// TIA Portal project "RedArrowMQTT" (V15)

(* hardware
DEVICE "S7-1200 station_1"  S7-1200 Station
   slot 0: "Rack_0"  S7-1200 Rack  Rack  V1.0
   slot 1: "PLC_1"  CPU 1214C AC/DC/Rly  6ES7 214-1BG40-0XB0  V4.2
*)

// ===== PLC "PLC_1"  CPU 1214C AC/DC/Rly =====

VAR_GLOBAL   // PLC tag table "Default tag table"
   "System_Byte" AT %MB1 : Byte;
   "FirstScan" AT %M1.0 : Bool;
   "DiagStatusUpdate" AT %M1.1 : Bool;
   "AlwaysTRUE" AT %M1.2 : Bool;
   "AlwaysFALSE" AT %M1.3 : Bool;
   "Clock_Byte" AT %MB0 : Byte;
   "Clock_10Hz" AT %M0.0 : Bool;
   "Clock_5Hz" AT %M0.1 : Bool;
   "Clock_2.5Hz" AT %M0.2 : Bool;
   "Clock_2Hz" AT %M0.3 : Bool;
   "Clock_1.25Hz" AT %M0.4 : Bool;
   "Clock_1Hz" AT %M0.5 : Bool;
   "Clock_0.625Hz" AT %M0.6 : Bool;
   "Clock_0.5Hz" AT %M0.7 : Bool;
   "miState" AT %MW50 : Int;
   "miCurrentLocation" AT %MW52 : Int;
   "SerializeResult" AT %MW56 : Int;
   "charCount" AT %MW54 : Int;
   "bSendMessage" AT %M35.0 : Bool;
   "bSubscribe" AT %M35.1 : Bool;
END_VAR

VAR_GLOBAL CONSTANT   // PLC tag table "IOT Constants"
   "ciSubMessageReceived" : Int := 15;
   "ciDisablePublish" : Int := 0;
   "ciSubReadyToSub" : Int := 10;
   "ciSubDisabled" : Int := 0;
   "ciSubSubscribed" : Int := 20;
   "ciReadyToPublish" : Int := 10;
END_VAR

VAR_GLOBAL CONSTANT   // PLC tag table "MQTT Message Constants"
   "ciRemovalRequested" : Int := 2;
   "ciAdditionRequested" : Int := 1;
   "ciDriverIDLength" : Int := 8;
   "ciVehicleIDLength" : Int := 8;
   "ciCustomerNameLength" : Int := 20;
   "ciMaxDrivers" : Int := 1000;
   "ciMaxVehicles" : Int := 1000;
   "ciMaxCustomers" : Int := 5;
   "ciWashesPerVehicle" : Int := 5;
   "ciSyncBufferSize" : Int := 75;
   "ciVersionNumber" : String := '/V3';
   "ciCustomerSyncBufferSize" : Int := 5;
END_VAR

TYPE "udtDriver"
   STRUCT
      sDriverID : String["ciDriverIDLength"];   // Driver's alphanumeric ID
      iCustomer : USInt;   // Index of customer to which driver belongs
   END_STRUCT;
END_TYPE

TYPE "udtVehicle"
   STRUCT
      sVehicleID : String["ciVehicleIDLength"];   // Vehicle ID
      iWashesAvailable : Array[1.."ciWashesPerVehicle"] of USInt;   // Set of wash types available to this vehicle
      iCustomer : USInt;   // Index of customer to which vehicle belongs
   END_STRUCT;
END_TYPE

TYPE "udtUserList"
   STRUCT
      Drivers : Array[1.."ciMaxDrivers"] of "udtDriver";
      Vehicles : Array[1.."ciMaxVehicles"] of "udtVehicle";
      Customers : Array[1.."ciMaxCustomers"] of String[20];
      sCurrentDriver : String["ciDriverIDLength"];
      sCurrentVehicleID : String["ciVehicleIDLength"];
      iCurrentWashesAvailable : Array[1.."ciWashesPerVehicle"] of USInt;
      iCurrentCustomer : USInt;
      sCurrentCustomerName : String["ciCustomerNameLength"];
   END_STRUCT;
END_TYPE

TYPE "udtError_Drivers"
   STRUCT
      DriverOverfill : Bool;   // Driver cannot be added because queue is full
      DriverDoesNotExist : Bool;   // Driver cannot be removed because they do not exist
      DriverExists : Bool;   // Driver cannot be added because they already exist
      CustomerDoesNotExist : Bool;   // Driver cannot be added or removed because customer does not exist
      SyncBufferOverfill : Bool;   // Sync operation cannot be completed due to lack of space
   END_STRUCT;
END_TYPE

TYPE "udtError_Vehicles"
   STRUCT
      VehicleOverfill : Bool;   // Vehicle cannot be added because queue is full
      VehicleDoesNotExist : Bool;   // Vehicle cannot be removed because they do not exist
      VehicleExists : Bool;   // Vehicle cannot be added because they already exist
      CustomerDoesNotExist : Bool;   // Vehicle cannot be added because customer does not exist
      SyncBufferOverfill : Bool;
   END_STRUCT;
END_TYPE

TYPE "udtError_Customer"
   STRUCT
      CustomerOverfill : Bool;   // Customer queue full
      CustomerAlreadyExists : Bool;   // Cannot add customer because they already exist
      CustomerDoesNotExist : Bool;   // Cannot remove custome because they do not exist
      SyncBufferOverfill : Bool;   // Customer sync buffer is full
   END_STRUCT;
END_TYPE

TYPE "udtCustomer"
   STRUCT
      sCustomerName : String["ciCustomerNameLength"];
      aVehicles : Array[1.."ciMaxVehicles"] of "udtVehicle";
      aDrivers : Array[1.."ciMaxDrivers"] of String["ciDriverIDLength"];
      Sync : Struct
         iTotalDrivers : Int;
         iTotalVehicles : Int;
         iDriversSynced : Int;   // Counter for how many drivers IDs have been sent so far suring the sync process
         iVehiclesSynced : Int;   // Counter for how many vehicles have been sent so far in the sync process
         sDriverSyncBuffer : Array[1.."ciSyncBufferSize"] of String[8];
         VehicleSyncBuffer : Array[1.."ciSyncBufferSize"] of "udtVehicle";
         bDriverSyncComplete : Bool;
         bVehicleSyncComplete : Bool;
         bDriverSync : Array[1.."ciMaxDrivers"] of Bool;   // Bit indicating if a driver at a given index has been synced
         bVehicleSync : Array[1.."ciMaxVehicles"] of Bool;   // Bit indicating if a vehicle at a given index has been synced
         bCustomerSync : Bool;
      END_STRUCT;
   END_STRUCT;
END_TYPE

TYPE "udtCustomerList"
   STRUCT
      aCustomers : Array[1.."ciMaxCustomers"] of "udtCustomer";
      sCurrentDriver : String["ciDriverIDLength"];
      sCurrentVehicleID : String["ciVehicleIDLength"];
      iCurrentWashesAvailable : Array[1.."ciWashesPerVehicle"] of USInt;
      iCurrentCustomer : USInt;
      sCurrentCustomerName : String["ciCustomerNameLength"];
      iTotalCustomers : Int;
      iCustomersSynced : Int;
   END_STRUCT;
END_TYPE

TYPE "udtWashReportRaw"
   STRUCT
      bInWashComplete : Bool := false;   // Trigger to start the serialization
      bInMaxRuntimeTripped : Bool;   // Set if the user wash in wash for more than max allowed time
      DTL_StartTime : DTL;   // Starting date and time of wash
      tInTotalTime : Time;   // Total time in wash
      iInWashType : USInt;   // Wash type ID
      tInArch1Time : Time;
      tInArch2Time : Time;
      tInArch3Time : Time;
      tInArch4Time : Time;
      tInArch5Time : Time;
   END_STRUCT;
END_TYPE

TYPE "udtWashReportSend"
   STRUCT
      sCustomer : String["ciCustomerNameLength"];   // Customer Name
      sDriverID : String["ciDriverIDLength"];   // 8 character alphanumeric driver ID
      sVehicleID : String["ciVehicleIDLength"];   // 8 character alphanumeric vehicle ID
      iWashType : UInt;   // Wash type received
      bInMaxRuntimeTripped : Bool;   // Set if the user wash in wash for more than max allowed time
      iYear : UInt;   // Year
      iMonth : UInt;   // Month
      iDay : UInt;   // Day
      iHour : UInt;   // Hour
      iMinute : UInt;   // Minute
      iSecond : UInt;   // Second
      iTotalTime : UInt;   // Total time in wash
      iArch1Time : UInt;   // Time under arch 1
      iArch2Time : UInt;   // Time under arch 2
      iArch3Time : UInt;   // Time under arch 3
      iArch4Time : UInt;   // Time under arch 4
      iArch5Time : UInt;   // Time under arch 5
   END_STRUCT;
END_TYPE

TYPE "udtSyncLog"
   STRUCT
      iTotalCustomers : UInt;
      iTotalDrivers : UInt;
      iTotalVehicles : UInt;
      iCustomersSynced : USInt;
      iVehiclesSynced : UInt;
      iDriversSynced : UInt;
      CustomerSyncBuffer : Array[1.."ciCustomerSyncBufferSize"] of String["ciCustomerNameLength"];
      DriverSyncBuffer : Array[1.."ciSyncBufferSize"] of "udtDriver";
      VehicleSyncBuffer : Array[1.."ciSyncBufferSize"] of "udtVehicle";
      bDriverSync : Array[1.."ciMaxDrivers"] of Bool;
      bVehicleSync : Array[1.."ciMaxVehicles"] of Bool;
      bCustomerSync : Array[1.."ciMaxCustomers"] of Bool;
   END_STRUCT;
END_TYPE

// folder: MQTT

TYPE "udtMQTT_SubcribeMessageBuffer"
   STRUCT
      Message : Array[1..20] of "udtMQTT_SubscribeMessage";   // udtMQTT_SubscribeMessage
   END_STRUCT;
END_TYPE

TYPE "udtMQTT_SubscribeMessage"
   STRUCT
      iStatus : Int;   // Message status
      iQoS : Int;   // Quality of service value (0 or 1)
      sTopic : String[75];   // Topic to which its subscribed
      byValue : Array[0..75] of Byte;   // Byte array of message contents
      iMessageLength : Int;   // Length of received message
   END_STRUCT;
END_TYPE

TYPE "udtMQTT_PublishMessage"
   STRUCT
      iStatus : Int;   // Message Status
      iQoS : Int;   // Quality of service value (0 or 1)
      sTopic : String;   // Topic of sent message
      byValue : Array[0..100] of Byte;   // Byte array of message contents
      iMessageLength : DInt;   // Length of byValue occupied by relevant data
   END_STRUCT;
END_TYPE

TYPE "udtMQTT_PublishMessageBuffer"
   STRUCT
      iIndexWrite : Int;   // Message index currently being written by an fcMQTT_SerializeMessage block
      iIndexMax : Int := 3;   // Max index writtable within the message array
      bErrorOverfill : Bool;   // Set when fcMQTT_SerializeMessage tries to write to an unsent message
      Message : Array[1..10] of "udtMQTT_PublishMessage";   // udtMQTT_PublishMessage
   END_STRUCT;
END_TYPE

TYPE "udtError_MQTT"
   STRUCT
      ConSendErr : Bool;
      ConSendTO : Bool;
      ConAckRcvErr : Bool;
      ConAckTO : Bool;
      ConAckIncReply : Bool;
      ConAckIncLen : Bool;
      ConAckUnacProt : Bool;
      ConAckIdRej : Bool;
      ConAckSerUn : Bool;
      ConAckUserPass : Bool;
      ConAckNotAut : Bool;
      ConAckUnknown : Bool;
      PubSendErr : Bool;
      PubSendTO : Bool;
      PubAckRcvErr : Bool;
      PubAckTO : Bool;
      PubAckIncReply : Bool;
      PubAckIncLen : Bool;
      PubAckPacketID : Bool;
      SubSendErr : Bool;
      SubSendTimeout : Bool;
      SubAckIncReply : Bool;
      SubAckPacketID : Bool;
      SubAckRcvErr : Bool;
      SubAckTO : Bool;
      SubTopicNotFound : Bool;
      SubSendPubAckErr : Bool;
      SubSendPubAckTO : Bool;
      TcpErr : Bool;
      TcpTO : Bool;
      QueueOverflow : Bool;
   END_STRUCT;
END_TYPE

// folder: (top level)

DATA_BLOCK "IOT Communication_DB"   // DB3
{ S7_Optimized_Access := 'TRUE' }
VERSION : 0.1
// stored: InstanceOfName IOT Communication
"IOT Communication"
BEGIN
END_DATA_BLOCK

DATA_BLOCK "fbMain_DB"   // DB4
{ S7_Optimized_Access := 'TRUE' }
VERSION : 0.1
// stored: InstanceOfName fbMain
"fbMain"
BEGIN
END_DATA_BLOCK

DATA_BLOCK "dbErrors"   // DB7
{ S7_Optimized_Access := 'TRUE' }
VERSION : 0.1
   VAR
      Error_MQTT : "udtError_MQTT";
      Error_Drivers : "udtError_Drivers";
      Error_Vehicles : "udtError_Vehicles";
      Error_Customers : "udtError_Customer";
   END_VAR
BEGIN
END_DATA_BLOCK

// folder: MQTT

DATA_BLOCK "dbMQTT_MessageBuffer"   // DB1
{ S7_Optimized_Access := 'TRUE' }
VERSION : 0.1
   VAR
      OutgoingMessages : "udtMQTT_PublishMessageBuffer";
      IncomingMessages : "udtMQTT_SubcribeMessageBuffer";
      ErrorMessages : "udtMQTT_PublishMessageBuffer";
   END_VAR
BEGIN
   OutgoingMessages.iIndexMax := 10;
   ErrorMessages.iIndexMax := 10;
   IncomingMessages.Message[1].iStatus := 0;
   IncomingMessages.Message[2].iStatus := 0;
   IncomingMessages.Message[3].iStatus := 0;
END_DATA_BLOCK

DATA_BLOCK "dbMQTT_Data"   // DB26
TITLE = gdbIOTData_V1
{ S7_Optimized_Access := 'FALSE' }
AUTHOR : Eric_Niebylski
VERSION : 0.1
// Added rTargetRate ro 10minDataorAlarm
   VAR
      TestTopic : Struct   // To IOT Only
         DeviceID : String[9] := 'Something';
      END_STRUCT;
      ConfigData : Struct   // Bi
         Param1 : Int;
         Param2 : Int;
         Param3 : Real;
      END_STRUCT;
      sTemp : String;
      testCharArray : Array[1..20] of Char;
      rTemp : Real;
      itemp : Int;
      wError : Word;
   END_VAR
BEGIN
END_DATA_BLOCK

// folder: System blocks/Program resources

DATA_BLOCK "MQTT_TCON_Param"   // DB2
{ S7_Optimized_Access := 'TRUE' }
AUTHOR : SIMATIC
FAMILY : MC7Plus
NAME : TCON_Prm
VERSION : 1.0
// stored: InstanceOfName TCON_Param
"TCON_Param"
BEGIN
   REM_TSAP_ID[1] := 16#07;
   REM_TSAP_ID[2] := 16#5B;
   ID := 4;
END_DATA_BLOCK

// folder: (top level)

FUNCTION_BLOCK "fbMain"   // FB1, LAD
{ S7_Optimized_Access := 'TRUE' }
VERSION : 0.1
   VAR
      ins_GET_IM_DATA : Get_IM_Data;
      IMData : IM0_Data;
      bIMDataDone : Bool;
      bReadyToSub : Bool;   // Ready to subscribe to topics
      insFb_TankLevel : "fbTankLevel";
      bInMid : Bool;
      bInLow : Bool;
      bValidDriver : Bool;
      bValidVehicle : Bool;
      "IOT Communication_DB" : "IOT Communication";
      bWashReportSend : Bool;
      TON_WashReportSend : TON_TIME;
   END_VAR
   VAR_TEMP
      iTemp1 : Int;
      diTemp : DInt;
      bTemp : Bool;
      wTemp : Word;
   END_VAR
BEGIN

REGION Network 1
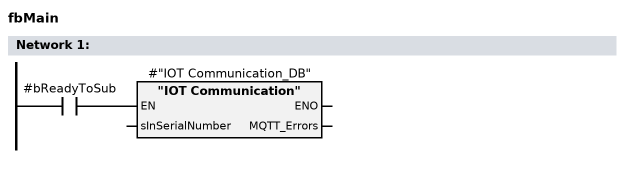
   RUNG wire#powerrail
      Contact( #bReadyToSub )
      #"IOT Communication_DB"(sInSerialNumber :=, MQTT_Errors =>)
   END_RUNG
   // the same network as SCL:
   IF #bReadyToSub THEN
       #"IOT Communication_DB"();   // "IOT Communication"
   END_IF;
END_REGION
END_FUNCTION_BLOCK

ORGANIZATION_BLOCK "Main"   // OB1, LAD, ProgramCycle
TITLE = "Main Program Sweep (Cycle)"
{ S7_Optimized_Access := 'TRUE' }
VERSION : 0.1
   VAR_INPUT
      Initial_Call : Bool;   // Initial call of this OB
      Remanence : Bool;   // =True, if remanent data are available
   END_VAR
BEGIN

REGION Network 1
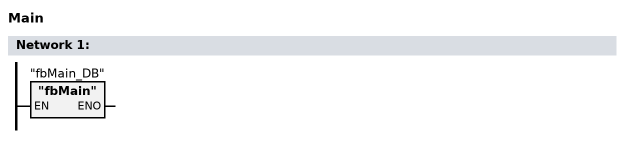
   RUNG wire#powerrail
      "fbMain_DB"()
   END_RUNG
   // the same network as SCL:
   "fbMain_DB"();   // "fbMain"
END_REGION
END_ORGANIZATION_BLOCK

// folder: MQTT

FUNCTION_BLOCK "IOT Communication"   // FB18, SCL
{ S7_Optimized_Access := 'TRUE' }
VERSION : 0.1
   VAR_INPUT
      sInSerialNumber : String;
   END_VAR
   VAR_OUTPUT
      MQTT_Errors : "udtError_MQTT";   // MQTT Error udt
   END_VAR
   VAR
      MQTT : "fbMQTT";
      bSerializeDone : Array[0..10] of Bool;
      bSerializeHold : Array[0..10] of Bool;
      bNewMessage : Array[0..10] of Bool;
      bInTankMidSensor : Bool;   // Temporary, replace with DI
      bInTankLowSensor : Bool;   // Temporary, replace with DI
      TankLevel : "fbTankLevel";
      bSendTankReport : Bool;
      iCustomersSynced : Int;
      sLastCustomerSync : String["ciCustomerNameLength"];
      sLastDriverSync : String["ciDriverIDLength"];
      sLastDriverCustomer : String["ciCustomerNameLength"];
      sLastVehicleSync : String["ciVehicleIDLength"];
      sLastVehicleCustomer : String["ciCustomerNameLength"];
   END_VAR
   VAR_TEMP
      tempTime : Time;
      bTemp : Bool;
      iIndex : Int;
      i : Int;
      diTemp : DInt;
   END_VAR
BEGIN
   // MQTT communication control driver
   #MQTT(sInClientID := 'ClientID',
         sInUserName := 'UserName',
                sInPassword := '12345',
                TCON_Param := "MQTT_TCON_Param",
                ERROR_MQTT := #MQTT_Errors);


    // Serialize message Structure to be sent
   "fcMQTT_SerializeMessageRaw"(sInSerial:=_string_in_,
                                sInTopic:=_string_in_,
                                sInVersion:=_string_in_,
                                iInQoS:=_int_in_,
                                Message:=_variant_in_,
                                bOutMessageSerialized=>_bool_out_);

   //Subscribe to message and send to DB
   "fcMQTT_DeserializeMessageSubscribe"(sInTopic:=_string_in_,
                                        iInQoS:=_int_in_,
                                        iInBufferIndex:=_int_in_,
                                        sInSerial:=_string_in_,
                                        sInVersion:=_string_in_,
                                        Message=>_variant_out_,
                                        bOutNewMessage=>_bool_out_);
END_FUNCTION_BLOCK

FUNCTION_BLOCK "fbMQTT"   // FB19, SCL
{ S7_Optimized_Access := 'TRUE' }
VERSION : 0.1
   VAR_INPUT
      sInClientID : String;   // Client ID, 23 char max / Client ID
      sInUserName : String;   // Username
      sInPassword : String;   // Password
      bInCleanSession : Bool;   // 0=Reuse prev session; 1=Discard prev sessions and start new one / Set high to clean session
      bInResetError : Bool;   // Error Reset
   END_VAR
   VAR_OUTPUT
      bOutError : Bool;   // Error present
   END_VAR
   VAR_IN_OUT
      ERROR_MQTT : "udtError_MQTT";   // Error udt
      TCON_Param : TCON_Param;   // Connection paramters
   END_VAR
   VAR
      iStatePublish : Int := 10;   // Current state of publish state machine
      iStateSubscribe : Int := 10;   // Current state of subscribe state machine
      iSelQueueIndexPublish : Int;   // Queue index of message currently being published
      iPrevSelQueueIndexPublish : Int;   // Queue index of last message to be published
      iPublishIndex : Int;   // Current byte index of message to be published
      uiSendLen : UInt;   // Length of message being sent
      uiPubPacketID : UInt;   // Unique ID for each sent packet
      bPubInProgress : Bool;   // Publication of packet in progress
      iSubscribeIndex : Int;   // Queue index of message whose topic is being subscribed to
      uiSubPacketID : UInt;   // ID of subcribe packet. Expected in suback packet.
      iSubMessageIndex : Int;   // Current byte of current working subscription related message
      bSubInProgress : Bool;   // Set if busy subscribing to a topic
      bSubReceiveInProgress : Bool;   // Set if busy receiving data on a subscribed topic
      iSubReceivedQoS : Int;   // QoS of received publish packet
      iReceivedTopicLength : Int;   // Length of a received topic (in bytes)
      sReceivedTopic : String;   // Topic of received message
      iTopicIndex : Int;   // Index of received topic within Incoming Messages
      bConAckReceived : Bool;   // Conack packet received
      bPubAckReceived : Bool;   // Puback packet received
      bSubAckReceived : Bool;   // Suback packet received
      bPublishReceived : Bool;   // Publish packet received
      iPayloadStartIndex : Int;   // Start index of payload of received publish packet
      iEndOfPayloadIndex : Int;   // End index of payload of received publish packet
      byData : Array[1..200] of Byte;   // Max: id+user+password+buffer
      byDataNewMessage : Array[1..300] of Byte;
      fbTCON : TCON;   // fb to establish TCP connection
      fbTDISCON : TDISCON;   // fb to disconnect from TCP
      fbTSEND : TSEND;   // fb for sending packets
      fbTRCV : TRCV;   // fb for receiving packets
      TON_TimeoutPub : TON_TIME;   // Publish timeout timer
      TON_TimeoutSub : TON_TIME;   // Subscribe timeout timer
      TON_DelaySubscribe : TON_TIME;   // To space out traffic, wait 5 seconds after MQTT connection to subscribe / Subscribe delay timer
      iNewDataIndex : Int := 1;   // Byte index of newly received packet
      bTCP_Connected : Bool;   // Set when TCP connection established
      bMQTT_Connected : Bool;   // Set when MQTT connection established
      iLen : Int;   // Length temp
      iStatePrevPub : Int;   // Previous publish state
      bStateTransitionPub : Bool;   // Set when publish state changes
      iStatePrevSub : Int;   // Previous subscribe state
      bStateTransitionSub : Bool;   // Set when subscribe state changes
      bReceiveMessageComplete : Bool;   // Set when a packet has been completely received
      iReceiveMessageLength : Int;   // Length of received packet
      iReceiveLengthCalcIndex : Int;   // Index wihtin received message header
      iErrIndex : Int := 1;   // Error index
   END_VAR
   VAR_TEMP
      byLSB : Byte;   // LSB of received packet ID
      byMSB : Byte;   // MSB of received packet ID
      wTemp : Word;   // Temp words used for finding received topic length
      wTemp2 : Word;
      wTemp3 : Word;
      wTemp4 : Word;
      i : Int;
      j : Int;
      iStartingIndex : Int;
      byTemp : Byte;
      uiTemp : UInt;
      uiTopicLen : UInt;
      multiplier : Int;
      byTopic : Array[0..100] of Byte;
      bTopicNotFound : Bool;   // Set until incoming message topic is found to match subscribed topic
   END_VAR
   VAR CONSTANT
      ciPubIdle : Int := 10;   // Publish idle state
      ciPubError : Int := 999;   // Publish error state
      ciEstablishTCP : Int := 100;   // TCP connection state
      ciPubConnect : Int := 20;   // MQTT connect packet creation state
      ciPubConnectSend : Int := 30;   // Connect packet sending state
      ciPubWaitConnack : Int := 40;   // Waiting for connack packet state
      ciPubPublish : Int := 50;   // Publish packet creation state
      ciPubSend : Int := 60;   // Publish packet sending state
      ciPubWaitPubAck : Int := 70;   // Waiting for puback packet state (if QoS = 1)
      ciPubRestart : Int := -1;   // Waiting to reenter PubIdle after an error state
      ciSubQueueSize : Int := 20;   // Total number of incoming message udts in buffer
      ciSubIdle : Int := 10;   // Subscribe idle state
      ciSubError : Int := 999;   // Subscribe error state
      ciSubSubscribe : Int := 30;   // Subscribe packet creation state
      ciSubSendSubscribe : Int := 40;   // Subscribe packet sending state
      ciSubWaitSuback : Int := 50;   // Waiting for suback packet state
      ciSubDataReceived : Int := 60;   // Decoding of publish packet for subscribed topic state
      ciSubSendPubAck : Int := 70;   // Puback packet creation state
   END_VAR
BEGIN
   //Publish state machine
   // Save previous state for use in timeout timer
   #iStatePrevPub := #iStatePublish;
   CASE #iStatePublish OF
       #ciPubIdle: // Check connections and scan for messages that are ready to send
           // Connect, by default, to TCP and MQTT
           IF NOT #bTCP_Connected THEN
               #iStatePublish := #ciEstablishTCP;
           END_IF;

           // Connect to MQTT once a TCP connection has been established
           IF #bTCP_Connected AND NOT #bMQTT_Connected THEN
               #iStatePublish := #ciPubConnect;
           END_IF;


           // If an element has already been selected to send, check that connections are established
           IF #iSelQueueIndexPublish > 0 THEN
               IF #bTCP_Connected AND #bMQTT_Connected AND #iStateSubscribe = #ciSubIdle THEN
                   // Only publish if connected and subscribe state machine is also idle
                   #iStatePublish := #ciPubPublish;
               END_IF;
           ELSE
               // Scan through elements in queue until finding one that's ready to send
               // Start scan at index after index of previously sent message to avoid bias towards sending low index elements
               FOR #i := 1 TO "dbMQTT_MessageBuffer".OutgoingMessages.iIndexMax DO
                   #j := #iPrevSelQueueIndexPublish + #i;
                   // Loop back to first index after exceeding max
                   IF (#j > "dbMQTT_MessageBuffer".OutgoingMessages.iIndexMax) THEN
                       #j := #j - "dbMQTT_MessageBuffer".OutgoingMessages.iIndexMax;
                   END_IF;
                   // Check if element is ready in the queue
                   IF ("dbMQTT_MessageBuffer".OutgoingMessages.Message[#j].iStatus = "ciReadyToPublish") THEN
                       #iSelQueueIndexPublish := #j;       // Record index of selected element
                       EXIT;
                   END_IF;
               END_FOR;
           END_IF;

       #ciPubConnect: // Send connect message
           ////////////////////////////////////
           // Create connect message
           ////////////////////////////////////

           //********* Configure Fixed Header ***********//
           #iPublishIndex := 1;
           #byData[#iPublishIndex] := 2#00010000;   // Packet type 0x1; Flags 0x0 (reserved)
           #iPublishIndex := #iPublishIndex + 1;

           //Reset all subscriptions
           FOR #i := 1 TO 20 BY 1 DO
               "dbMQTT_MessageBuffer".IncomingMessages.Message[#i].iStatus := "ciSubDisabled";
           END_FOR;

           // Calculate remaining length (see MQTT doc)
           #iLen := 12 + LEN(#sInClientID);
           IF LEN(#sInUserName) > 0 THEN
               #iLen := #iLen + LEN(#sInUserName) + 2;
           END_IF;
           IF LEN(#sInPassword) > 0 THEN
               #iLen := #iLen + LEN(#sInPassword) + 2;
           END_IF;
           REPEAT
               #byTemp := INT_TO_BYTE(#iLen MOD 128);
               #iLen := #iLen / 128;
               // If there is more data to encode, set bit 7 high
               IF #iLen > 0 THEN
                   #byTemp := #byTemp OR 2#10000000;
               END_IF;
               #byData[#iPublishIndex] := #byTemp;
               #iPublishIndex := #iPublishIndex + 1;
           UNTIL #iLen <= 0 END_REPEAT;

           //********* Variable Header ***********//
           #byData[#iPublishIndex] := 16#00;    // Length MSB
           #iPublishIndex := #iPublishIndex + 1;
           #byData[#iPublishIndex] := 16#04;    // Length LSB
           #iPublishIndex := #iPublishIndex + 1;
           #byData[#iPublishIndex] := CHAR_TO_BYTE('M');
           #iPublishIndex := #iPublishIndex + 1;
           #byData[#iPublishIndex] := CHAR_TO_BYTE('Q');
           #iPublishIndex := #iPublishIndex + 1;
           #byData[#iPublishIndex] := CHAR_TO_BYTE('T');
           #iPublishIndex := #iPublishIndex + 1;
           #byData[#iPublishIndex] := CHAR_TO_BYTE('T');
           #iPublishIndex := #iPublishIndex + 1;
           #byData[#iPublishIndex] := 16#04;     // Protocol level 0x04
           #iPublishIndex := #iPublishIndex + 1;

           // Build connect flags, ignoring will message
           #byData[#iPublishIndex] := 16#00;       // Initialize with no flags set
           IF LEN(#sInUserName) > 0 THEN
               #byData[#iPublishIndex] := #byData[#iPublishIndex] OR 2#10000000;
           END_IF;
           IF LEN(#sInPassword) > 0 THEN
               #byData[#iPublishIndex] := #byData[#iPublishIndex] OR 2#01000000;
           END_IF;
           IF #bInCleanSession THEN
               #byData[#iPublishIndex] := #byData[#iPublishIndex] OR 2#00000010;
           END_IF;
           #iPublishIndex := #iPublishIndex + 1;
           #byData[#iPublishIndex] := 16#0E;  // Keepalive MSB, in seconds
           #iPublishIndex := #iPublishIndex + 1;
           #byData[#iPublishIndex] := 16#10;  // Keepalive LSB, in seconds
           #iPublishIndex := #iPublishIndex + 1;

           // Payload - client ID
           #iLen := LEN(#sInClientID);
           // Convert length int to a word and bit shift right to isolate MSB
           #byData[#iPublishIndex] := WORD_TO_BYTE(SHR(IN := INT_TO_WORD(#iLen), N := 8));   // String length MSB
           #iPublishIndex := #iPublishIndex + 1;
           // Convert length int to a word and drive bits 8-15 to 0 to isolate LSB
           #byData[#iPublishIndex] := WORD_TO_BYTE(INT_TO_WORD(#iLen) AND 16#00FF);   // String length LSB            
           #iPublishIndex := #iPublishIndex + 1;
           // Copy sInClientID into byData
           FOR #i := 1 TO #iLen DO
               #byData[#iPublishIndex] := CHAR_TO_BYTE(#sInClientID[#i]);
               #iPublishIndex := #iPublishIndex + 1;
           END_FOR;

           // Payload - User name
           IF LEN(#sInUserName) > 0 THEN
               #iLen := LEN(#sInUserName);
               // Convert length int to a word and bit shift right to isolate MSB
               #byData[#iPublishIndex] := WORD_TO_BYTE(SHR(IN := INT_TO_WORD(#iLen), N := 8));   // String lenght MSB
               #iPublishIndex := #iPublishIndex + 1;
               // Convert length int to a word and drive bits 8-15 to 0 to isolate LSB
               #byData[#iPublishIndex] := WORD_TO_BYTE(INT_TO_WORD(#iLen) AND 16#00FF);   // String lenght LSB            
               #iPublishIndex := #iPublishIndex + 1;
               // Copy sInUserName into byData
               FOR #i := 1 TO #iLen DO
                   #byData[#iPublishIndex] := CHAR_TO_BYTE(#sInUserName[#i]);
                   #iPublishIndex := #iPublishIndex + 1;
               END_FOR;
           END_IF;

           // Payload - password
           IF LEN(#sInPassword) > 0 THEN
               #iLen := LEN(#sInPassword);
               // Convert length int to a word and bit shift right to isolate MSB
               #byData[#iPublishIndex] := WORD_TO_BYTE(SHR(IN := INT_TO_WORD(#iLen), N := 8));   // String lenght MSB
               #iPublishIndex := #iPublishIndex + 1;
               // Convert length int to a word and drive bits 8-15 to 0 to isolate LSB
               #byData[#iPublishIndex] := WORD_TO_BYTE(INT_TO_WORD(#iLen) AND 16#00FF);   // String lenght LSB            
               #iPublishIndex := #iPublishIndex + 1;
               // Copy sInPassword into byData
               FOR #i := 1 TO #iLen DO
                   #byData[#iPublishIndex] := CHAR_TO_BYTE(#sInPassword[#i]);
                   #iPublishIndex := #iPublishIndex + 1;
               END_FOR;
           END_IF;

           //********* Send Packet ***********//
           #uiSendLen := INT_TO_UINT(#iPublishIndex - 1);   // Update packet length
           #iStatePublish := #ciPubConnectSend;  // Send packet packet

       #ciPubConnectSend:
           IF #fbTSEND.DONE THEN
               // All good. Receive Connack message
               #iStatePublish := #ciPubWaitConnack;
           ELSIF #fbTSEND.ERROR THEN
               // Sending error
               #ERROR_MQTT.ConSendErr := true;
               #iStatePublish := #ciPubError;
           ELSIF #TON_TimeoutPub.Q THEN
               // Timeout error
               #ERROR_MQTT.ConSendTO := true;
               #iStatePublish := #ciPubError;
           END_IF;

       #ciPubWaitConnack:
           ////////////////////////////////////
           // Process connection acknowledgement message
           ////////////////////////////////////
           IF #bConAckReceived THEN
               //Reset received flag
               #bConAckReceived := FALSE;
               // Parse received data
               // Header should be 0x20
               IF #byDataNewMessage[1] <> 16#20 THEN
                   #ERROR_MQTT.ConAckIncReply := true;
                   #iStatePublish := #ciPubError;
                   // Remaining length should be 2
               ELSIF #byDataNewMessage[2] <> 2 THEN
                   #ERROR_MQTT.ConAckIncLen := true;
                   #iStatePublish := #ciPubError;
                   // TODO: Parse SP flag?
                   // Return code should be 0    
               ELSIF #byDataNewMessage[4] <> 0 THEN
                   // Parse error code
                   IF #byDataNewMessage[4] = 1 THEN
                       // Connection refused, unaccepted protocol version
                       #ERROR_MQTT.ConAckUnacProt := TRUE;
                   ELSIF #byDataNewMessage[4] = 2 THEN
                       // Connection refused, identifier rejected
                       #ERROR_MQTT.ConAckIdRej := TRUE;
                   ELSIF #byDataNewMessage[4] = 3 THEN
                       // Connection refused, server unavailable
                       #ERROR_MQTT.ConAckSerUn := TRUE;
                   ELSIF #byDataNewMessage[4] = 4 THEN
                       // Connection refused, bad username or password
                       #ERROR_MQTT.ConAckUserPass := TRUE;
                   ELSIF #byDataNewMessage[4] = 5 THEN
                       // Connection refused, client not authorized to connect
                       #ERROR_MQTT.ConAckNotAut := TRUE;
                   ELSE
                       // Error unknown
                       #ERROR_MQTT.ConAckUnknown := TRUE;
                   END_IF;
                   #iStatePublish := #ciPubError;
               ELSE
                   // Everything is correct and a connection has been established
                   #bMQTT_Connected := true;
                   #iStatePublish := #ciPubIdle;
               END_IF;
           (*ELSIF #fbTRCV.ERROR THEN
               // Receive error
               #ERROR_MQTT.ConAckRcvErr := true;
               "dbTestingJJC".wDisError := #fbTRCV.STATUS;
               #iStatePublish := #ciPubError;*)
           ELSIF #TON_TimeoutPub.Q THEN
               #ERROR_MQTT.ConAckTO := true;
               #iStatePublish := #ciPubError;
           END_IF;

       #ciPubPublish:
           ////////////////////////////////////
           // Create publish message
           ////////////////////////////////////

           //********* Configure Fixed Header ***********//
           #iPublishIndex := 1;    // Reset index to 1 for creation of new message
           #byData[#iPublishIndex] := 2#00110000;   // Packet type 0x3;
           IF #bPubInProgress THEN
               #byData[#iPublishIndex] := #byData[#iPublishIndex] OR 2#00001000; // DUP flag. Re-delivery attempt
           ELSE
               // New send attempt - Increment Packet ID
               #uiPubPacketID := #uiPubPacketID + 1;
           END_IF;

           // QoS flag, assuming 0 by default
           IF "dbMQTT_MessageBuffer".OutgoingMessages.Message[#iSelQueueIndexPublish].iQoS = 1 THEN
               #byData[#iPublishIndex] := #byData[#iPublishIndex] OR 2#00000010; // QoS flag
           END_IF;
           //TODO: QoS 2 is not currently implemented by adafruit
           // TODO: Ignoring retain flag for now
           #iPublishIndex := #iPublishIndex + 1;

           // Calculate remaining length (see MQTT doc)
           #iLen := LEN("dbMQTT_MessageBuffer".OutgoingMessages.Message[#iSelQueueIndexPublish].sTopic) + 2 + DINT_TO_INT("dbMQTT_MessageBuffer".OutgoingMessages.Message[#iSelQueueIndexPublish].iMessageLength);
           IF "dbMQTT_MessageBuffer".OutgoingMessages.Message[#iSelQueueIndexPublish].iQoS > 0 THEN
               // Adding packet ID for QoS 1 and 2
               #iLen := #iLen + 2;
           END_IF;

           REPEAT
               #byTemp := INT_TO_BYTE(#iLen MOD 128);
               #iLen := #iLen / 128;
               // If there is more data to encode then set bit 7 of the byte to 1
               IF #iLen > 0 THEN
                   #byTemp := #byTemp OR 2#10000000;
               END_IF;
               #byData[#iPublishIndex] := #byTemp;
               #iPublishIndex := #iPublishIndex + 1;
           UNTIL #iLen <= 0 END_REPEAT;

           //********* Variable Header ***********//
           // Topic name
           // The first and second bytes are the MSB and LSB (respectively) of the topic length 
           #iLen := LEN("dbMQTT_MessageBuffer".OutgoingMessages.Message[#iSelQueueIndexPublish].sTopic);
           #byData[#iPublishIndex] := WORD_TO_BYTE(SHR(IN := INT_TO_WORD(#iLen), N := 8));   // String length MSB
           #iPublishIndex := #iPublishIndex + 1;
           #byData[#iPublishIndex] := WORD_TO_BYTE(INT_TO_WORD(#iLen) AND 16#00FF);   // String length LSB
           #iPublishIndex := #iPublishIndex + 1;
           // Copy the topic name into the variable header
           FOR #i := 1 TO #iLen DO
               #byData[#iPublishIndex] := CHAR_TO_BYTE("dbMQTT_MessageBuffer".OutgoingMessages.Message[#iSelQueueIndexPublish].sTopic[#i]);
               #iPublishIndex := #iPublishIndex + 1;
           END_FOR;
           // Packet ID
           // If QoS > 0 then the variable header needs to include 2 bytes to act as an identifier for the packet
           IF "dbMQTT_MessageBuffer".OutgoingMessages.Message[#iSelQueueIndexPublish].iQoS > 0 THEN
               #byData[#iPublishIndex] := WORD_TO_BYTE(SHR(IN := UINT_TO_WORD(#uiPubPacketID), N := 8));   // Packet ID MSB
               #iPublishIndex := #iPublishIndex + 1;
               #byData[#iPublishIndex] := WORD_TO_BYTE(UINT_TO_WORD(#uiPubPacketID) AND 16#00FF);   // PacketID LSB
               #iPublishIndex := #iPublishIndex + 1;
           END_IF;

           //********* Payload ***********//
           // Assuming strings, without string length
           // According to the spec, server should calculate the length of the payload
           #iLen := DINT_TO_INT("dbMQTT_MessageBuffer".OutgoingMessages.Message[#iSelQueueIndexPublish].iMessageLength);
           FOR #i := 0 TO #iLen - 1 DO
               // Copy message into packet payload
               #byData[#iPublishIndex] := "dbMQTT_MessageBuffer".OutgoingMessages.Message[#iSelQueueIndexPublish].byValue[#i];
               #iPublishIndex := #iPublishIndex + 1;
           END_FOR;

           // Send message
           #bPubInProgress := true;
           #uiSendLen := INT_TO_UINT(#iPublishIndex - 1);   // Update packet length
           #iStatePublish := #ciPubSend;

       #ciPubSend:
           IF #fbTSEND.DONE THEN
               // QoS=1: Should receive puback message
               IF "dbMQTT_MessageBuffer".OutgoingMessages.Message[#iSelQueueIndexPublish].iQoS = 1 THEN
                   #iStatePublish := #ciPubWaitPubAck;
               ELSE
                   // QoS=0; No response from the server
                   // Remove message from the queue
                   "dbMQTT_MessageBuffer".OutgoingMessages.Message[#iSelQueueIndexPublish].iStatus := "ciDisablePublish";
                   #iPrevSelQueueIndexPublish := #iSelQueueIndexPublish;   // Save previous queue position
                   #iSelQueueIndexPublish := 0;                            // Reset queue position
                   #bPubInProgress := false;                               // Reset flag
                   #iStatePublish := #ciPubIdle;                           // Return to idle
               END_IF;
               // TODO: Handle QoS 2?
           ELSIF #fbTSEND.ERROR THEN
               // Send error
               #ERROR_MQTT.PubSendErr := true;
               #iStatePublish := #ciPubError;
           ELSIF #TON_TimeoutPub.Q THEN
               // Timeout error
               #ERROR_MQTT.PubSendTO := true;
               #iStatePublish := #ciPubError;
           END_IF;

       #ciEstablishTCP:
           // Wait for done or error flag
           IF #fbTCON.DONE THEN
               // TCP connection established 
               #bTCP_Connected := true;
               #bMQTT_Connected := false;
               #iStatePublish := #ciPubConnect;
           ELSIF #fbTCON.ERROR THEN
               "dbMQTT_Data".wError := #fbTCON.STATUS;
               // Connection failed
               #ERROR_MQTT.TcpErr := true;
               IF #fbTCON.STATUS = 16#80A3 THEN
                   // ID is used by a connection created by the user program,
                   // which uses the same connection description at the CONNECT parameter
                   #TCON_Param.ID := #TCON_Param.ID + 1;
               END_IF;
               IF #TCON_Param.ID > 9 THEN
                   #TCON_Param.ID := 1;
               END_IF;
               #iStatePublish := #ciPubError;
           ELSIF #TON_TimeoutPub.Q THEN
               // Timeout error
               #ERROR_MQTT.TcpTO := true;
               #iStatePublish := #ciPubError;
           END_IF;

       #ciPubWaitPubAck:
           IF #bPubAckReceived THEN
               #bPubAckReceived := false;
               // Parse received data
               // Header should be 0x40
               IF #byDataNewMessage[2] <> 16#02 THEN
                   // PubAck message should have a remaining length of 2
                   // TODO pub ack length error
                   #iStatePublish := #ciPubError;
               ELSE
                   // Check that the variable header matches the ID of the sent packet
                   #uiTemp := WORD_TO_UINT(SHL(IN := BYTE_TO_WORD(#byDataNewMessage[3]), N := 8) + BYTE_TO_WORD(#byDataNewMessage[4]));
                   IF #uiTemp <> #uiPubPacketID THEN
                       // Incorrect packet ID
                       #ERROR_MQTT.PubAckPacketID := TRUE;
                       #iStatePublish := #ciPubError;
                   ELSE
                       // All good. Reset queue and restart
                       "dbMQTT_MessageBuffer".OutgoingMessages.Message[#iSelQueueIndexPublish].iStatus := "ciDisablePublish";
                       #iPrevSelQueueIndexPublish := #iSelQueueIndexPublish;   // Save previous queue position
                       #iSelQueueIndexPublish := 0;                            // Reset queue position
                       #bPubInProgress := false;                               // Reset flag
                       #iStatePublish := #ciPubIdle;                           // Return to idle
                   END_IF;
               END_IF;
           ELSIF #fbTRCV.ERROR THEN
               // Receive error
               #ERROR_MQTT.PubAckRcvErr := TRUE;
               #iStatePublish := #ciPubError;
           ELSIF #TON_TimeoutPub.Q THEN
               // Timeout error
               #ERROR_MQTT.PubAckTO := true;
               #iStatePublish := #ciPubError;
           END_IF;

       #ciPubError:
           // Reset TCP connection
           #bMQTT_Connected := false;
           #bTCP_Connected := false;
           IF #fbTDISCON.DONE THEN
               #iStatePublish := #ciPubRestart;
           ELSIF #TON_TimeoutPub.Q THEN
               // Already wait for timeout, just jump to idle
               #iStatePublish := #ciPubIdle;
               #iNewDataIndex := 1;
           END_IF;

       #ciPubRestart:
           // Wait before restarting after the error
           IF #TON_TimeoutPub.Q THEN
               // Restart from IDLE
               #iStatePublish := #ciPubIdle;
               #iNewDataIndex := 1;
           END_IF;

       ELSE
           #iStatePublish := #ciPubIdle;

   END_CASE;

   // Timeout timer
   #bStateTransitionPub := #iStatePublish <> #iStatePrevPub;
   #TON_TimeoutPub(IN := ((NOT #bStateTransitionPub) AND (#iStatePublish <> #ciPubIdle)), PT := T#20S);

   // Subscribe state machine
   #iStatePrevSub := #iStateSubscribe;
   CASE #iStateSubscribe OF
       #ciSubIdle:
           #bSubInProgress := false;
           #bSubReceiveInProgress := false;
           // Wait until TCP and MQTT connected
           IF #TON_DelaySubscribe.Q THEN
               // Check if any new data has arrived
               IF #bPublishReceived THEN
                   // Reset flag
                   #bPublishReceived := false;
                   // If data has arrived, move to data received state
                   #iStateSubscribe := #ciSubDataReceived;
                   // Set flag to prevent sending other messages out
                   #bSubReceiveInProgress := true;
               END_IF;

               // Check for any unsubscribed topics
               IF NOT #bSubReceiveInProgress THEN
                   FOR #i := 1 TO #ciSubQueueSize BY 1 DO
                       IF "dbMQTT_MessageBuffer".IncomingMessages.Message[#i].iStatus = "ciSubReadyToSub" THEN
                           //If unsubscribed topic found, move to sub state and stop looking for new topics
                           #iStateSubscribe := #ciSubSubscribe;
                           #iSubscribeIndex := #i;
                           #bSubInProgress := true;
                           EXIT;
                       END_IF;
                   END_FOR;
               END_IF;
           END_IF;

       #ciSubSubscribe:
           //create subscribe MQTT packet
           #i := 1;
           #iSubMessageIndex := 1;
           #byData[#iSubMessageIndex] := 2#10000010;   // Packet type 0x80; Flags 0x02 (reserved)
           #iSubMessageIndex := #iSubMessageIndex + 1;

           // Calculate remaining length (see MQTT doc)
           // packet identifier (2) + topic length (2) + topic ( + QoS (1)
           #iLen := LEN("dbMQTT_MessageBuffer".IncomingMessages.Message[#iSubscribeIndex].sTopic) + 5;
           //Create encoding for packet length
           REPEAT
               #byTemp := INT_TO_BYTE(#iLen MOD 128);
               #iLen := #iLen / 128;
               // If there's more data to encode set bit 7 to 1
               IF #iLen > 0 THEN
                   #byTemp := #byTemp OR 2#10000000;
               END_IF;
               #byData[#iSubMessageIndex] := #byTemp;
               #iSubMessageIndex := #iSubMessageIndex + 1;
           UNTIL #iLen <= 0 END_REPEAT;

           // Increment packet ID and encode into variable header
           #uiSubPacketID := #uiSubPacketID + 1;
           // Bit shift uiSubPacketID 8 bits to the right to isolate the MSB 
           #byData[#iSubMessageIndex] := WORD_TO_BYTE(SHR(IN := UINT_TO_WORD(#uiSubPacketID), N := 8));   // Packet ID MSB
           #iSubMessageIndex := #iSubMessageIndex + 1;
           // Reset bits 8-15 of uiSubPacketID to isolate the LSB
           #byData[#iSubMessageIndex] := WORD_TO_BYTE(UINT_TO_WORD(#uiSubPacketID) AND 16#00FF);   // PacketID LSB
           #iSubMessageIndex := #iSubMessageIndex + 1;

           // Build payload
           // Only 1 topic. 2 bytes for length, topic, 1 byte for QoS
           // Length
           #uiTopicLen := INT_TO_UINT(LEN("dbMQTT_MessageBuffer".IncomingMessages.Message[#iSubscribeIndex].sTopic));
           // Bit shift uiTopicLen 8 bits to the right to isolate the MSB 
           #byData[#iSubMessageIndex] := WORD_TO_BYTE(SHR(IN := UINT_TO_WORD(#uiTopicLen), N := 8));   // Packet ID MSB
           #iSubMessageIndex := #iSubMessageIndex + 1;
           // Reset bits 8-15 of uiTopicLen to isolate the LSB
           #byData[#iSubMessageIndex] := WORD_TO_BYTE(UINT_TO_WORD(#uiTopicLen) AND 16#00FF);   // PacketID LSB
           #iSubMessageIndex := #iSubMessageIndex + 1;

           // Topic name
           #iLen := LEN("dbMQTT_MessageBuffer".IncomingMessages.Message[#iSubscribeIndex].sTopic);
           // Copy each character from the topic name into the payload
           FOR #i := 1 TO #iLen DO
               #byData[#iSubMessageIndex] := CHAR_TO_BYTE("dbMQTT_MessageBuffer".IncomingMessages.Message[#iSubscribeIndex].sTopic[#i]);
               #iSubMessageIndex := #iSubMessageIndex + 1;
           END_FOR;

           //QoS
           IF "dbMQTT_MessageBuffer".IncomingMessages.Message[#iSubscribeIndex].iQoS = 1 THEN
               #byData[#iSubMessageIndex] := 2#00000001;
           ELSE
               #byData[#iSubMessageIndex] := 2#00000000;
           END_IF;
           #uiSendLen := INT_TO_UINT(#iSubMessageIndex);
           #iStateSubscribe := #ciSubSendSubscribe;

       #ciSubSendSubscribe:
           IF #fbTSEND.DONE THEN
               #iStateSubscribe := #ciSubWaitSuback;

               IF "dbMQTT_MessageBuffer".IncomingMessages.Message[#iSubscribeIndex].iQoS = 0 THEN
                   #iStateSubscribe := #ciSubWaitSuback;
               END_IF;
           ELSIF #fbTSEND.ERROR THEN
               // Send error
               #ERROR_MQTT.PubSendErr := true;
               #iStateSubscribe := #ciPubError;
           ELSIF #TON_TimeoutSub.Q THEN
               // Timeout error
               #ERROR_MQTT.PubSendTO := true;
               #iStateSubscribe := #ciPubError;
           END_IF;

       #ciSubWaitSuback:
           //validate packet received. Should have same packet ID
           //
           IF #bSubAckReceived THEN
               #bSubAckReceived := false;
               // Parse received data
               // We know that we got an expected length
               // Header should be 0x90
               // Variable header = message id
               #uiTemp := WORD_TO_UINT(SHL(IN := BYTE_TO_WORD(#byDataNewMessage[3]), N := 8) + BYTE_TO_WORD(#byDataNewMessage[4]));

               IF #uiTemp <> #uiSubPacketID THEN
                   // Incorerct packet ID
                   #ERROR_MQTT.SubAckPacketID := TRUE;
                   #iStateSubscribe := #ciSubError;
                   //TODO also check QoS?
               ELSE
                   // All good. Reset queue and restart
                   "dbMQTT_MessageBuffer".IncomingMessages.Message[#iSubscribeIndex].iStatus := "ciSubSubscribed";
                   #iStateSubscribe := #ciSubIdle;
               END_IF;
           (* ELSIF #fbTRCV.ERROR THEN
               // Receive error
               #ERROR_MQTT.SubAckRcvErr := TRUE;
               #iStateSubscribe := #ciSubError; *)
           ELSIF #TON_TimeoutSub.Q THEN
               // Timeout error
               #ERROR_MQTT.SubAckTO := true;
               #iStateSubscribe := #ciSubError;
           END_IF;


       #ciSubDataReceived:
           // Reset flag
           #bSubReceiveInProgress := false;
           //find QoS
           #iSubMessageIndex := 1;
           #iSubReceivedQoS := 0;
           //TODO handling for QoS 2
           // Check for QoS 1 flag
           IF (#byDataNewMessage[#iSubMessageIndex] AND 2#00000010) = 2#00000010 THEN
               #iSubReceivedQoS := 1;
           END_IF;

           // Calculate message length
           #multiplier := 1;
           #iLen := 0;
           #iSubMessageIndex := 2;
           // Decode remaining length in accordance with MQTT doc
           REPEAT
               #byTemp := #byDataNewMessage[#iSubMessageIndex];
               #iLen := #iLen + (#byTemp AND 127) * #multiplier;
               #multiplier := #multiplier * 128;
               //TODO implement exception for length error
               #iSubMessageIndex := #iSubMessageIndex + 1;
           UNTIL ((#byTemp AND 128) = 0) END_REPEAT;

           // Find end index of message
           #iEndOfPayloadIndex := #iLen + #iSubMessageIndex - 1;

           // Find topic name
           // Find topic length
           #wTemp := 16#0000;
           #wTemp2 := 16#0000;
           #wTemp := #wTemp OR #byDataNewMessage[#iSubMessageIndex];   // Topic Length MSB
           #iSubMessageIndex := #iSubMessageIndex + 1;
           #wTemp2 := #byDataNewMessage[#iSubMessageIndex];            // Topic length LSB
           #wTemp3 := SHL(IN := #wTemp, N := 8);       // Bit shift MSB
           #wTemp4 := #wTemp OR #wTemp2;       // Combine MSB and LSB to get topic length 
           #iReceivedTopicLength := WORD_TO_INT(IN := #wTemp4);    // Convert to int
           #iSubMessageIndex := #iSubMessageIndex + 1;
           #iStartingIndex := #iSubMessageIndex;       // First index in topic name
           #j := 0;
           // Loop through message and copy in topic
           FOR #i := #iStartingIndex TO #iStartingIndex + #iReceivedTopicLength - 1 BY 1 DO
               #byTopic[#j] := #byDataNewMessage[#iSubMessageIndex];
               #j := #j + 1;
               #iSubMessageIndex := #iSubMessageIndex + 1;
           END_FOR;

           Chars_TO_Strg(Chars:=#byTopic, pChars:=0, Cnt:=INT_TO_UINT(#iReceivedTopicLength), Strg=>#sReceivedTopic);
           // Find index of topic
           #bTopicNotFound := TRUE;
           FOR #i := 1 TO #ciSubQueueSize BY 1 DO
               IF ("dbMQTT_MessageBuffer".IncomingMessages.Message[#i].sTopic = #sReceivedTopic) THEN
                   #iTopicIndex := #i;
                   #bTopicNotFound := FALSE;
                   EXIT;
               END_IF;
           END_FOR;

           //Throw error if topic not found
           IF #bTopicNotFound THEN
               #ERROR_MQTT.SubTopicNotFound := TRUE;
               #iStatePrevSub := #ciSubError;
           END_IF;

           //Depending on QoS go to idle or send PubAck reply
           IF (#iSubReceivedQoS = 0) THEN
               #iStateSubscribe := #ciSubIdle;
           ELSIF (#iSubReceivedQoS = 1) THEN

               //Find packet ID
               #byMSB := #byDataNewMessage[#iSubMessageIndex];
               #iSubMessageIndex := #iSubMessageIndex + 1;
               #byLSB := #byDataNewMessage[#iSubMessageIndex];
               #iSubMessageIndex := #iSubMessageIndex + 1;

               //build reply message
               //Control packet 16#40
               #byData[1] := 16#40;
               //remaining length is 2
               #byData[2] := 16#02;
               //add packet id
               #byData[3] := #byMSB;
               #byData[4] := #byLSB;
               #uiSendLen := 4;

               #iStateSubscribe := #ciSubSendPubAck;
           END_IF;

           // Get message
           IF NOT #bTopicNotFound THEN
               #iPayloadStartIndex := #iSubMessageIndex;
               #j := 0;
               FOR #i := #iPayloadStartIndex TO #iEndOfPayloadIndex BY 1 DO
                   // Copy the message into the incoming message space
                   "dbMQTT_MessageBuffer".IncomingMessages.Message[#iTopicIndex].byValue[#j] := #byDataNewMessage[#i];
                   #j := #j + 1;
               END_FOR;

               // Move topic and payload into received queue and set status
               "dbMQTT_MessageBuffer".IncomingMessages.Message[#iTopicIndex].iStatus := "ciSubMessageReceived";
               "dbMQTT_MessageBuffer".IncomingMessages.Message[#iTopicIndex].iMessageLength := #j;
           END_IF;

       #ciSubSendPubAck:
           IF #fbTSEND.DONE THEN
               #iStateSubscribe := #ciSubIdle;
           ELSIF #fbTSEND.ERROR THEN
               // Send error
               #ERROR_MQTT.SubSendPubAckErr := true;
               #iStateSubscribe := #ciPubError;
           ELSIF #TON_TimeoutSub.Q THEN
               #ERROR_MQTT.SubSendPubAckTO := true;
               #iStateSubscribe := #ciPubError;
           END_IF;

       #ciSubError:
           // Reset TCP connection
           #bMQTT_Connected := false;
           #bTCP_Connected := false;
           IF #fbTDISCON.DONE OR #fbTDISCON.ERROR THEN
               #iStateSubscribe := #ciPubRestart;
           ELSIF #TON_TimeoutSub.Q THEN
               // Already wait for timeout, just jump to idle
               #iStateSubscribe := #ciSubIdle;
           END_IF;

       #ciPubRestart:
           // Wait before restarting after the error
           IF #TON_TimeoutSub.Q THEN
               // Restart from IDLE
               #iStateSubscribe := #ciSubIdle;
           END_IF;


       ELSE
           #iStateSubscribe := #ciSubIdle;

   END_CASE;

   // Timeoout timer
   #bStateTransitionSub := #iStateSubscribe <> #iStatePrevSub;
   #TON_TimeoutSub(IN := ((NOT #bStateTransitionSub) AND (#iStateSubscribe <> #ciSubIdle)),
                   PT := T#20S);

   #TON_DelaySubscribe(IN := #bMQTT_Connected,
                       PT := T#3S);


   //Receive TCP data AND set flags
   IF #bReceiveMessageComplete AND #iNewDataIndex > 0 THEN

       // ConnAck Header 1st Byte: 00100000
       IF #byDataNewMessage[1] = 16#20 THEN
           #bConAckReceived := TRUE;
       END_IF;

       // PubAck Header 1st Byte: 01000000 
       IF #byDataNewMessage[1] = 16#40 THEN
           #bPubAckReceived := TRUE;
       END_IF;

       // SubAck Header 1st Byte: 10010000
       IF #byDataNewMessage[1] = 16#90 THEN
           #bSubAckReceived := TRUE;
       END_IF;

       // Publish Header 1st Byte: 0011XXXX
       IF (#byDataNewMessage[1] AND 2#11110000) = 16#30 AND #iStateSubscribe = #ciSubIdle THEN
           #bPublishReceived := TRUE;
       END_IF;

       #iNewDataIndex := 1;        // Reset iNewDataIndex to 1 to allow next message to be properly received

       #bReceiveMessageComplete := FALSE;      // Reset flag
       #iReceiveMessageLength := 0;            // Reset iReceiveMessageLength parameter


   END_IF;



   //**********************************************************************************************************************
   // Communicaiton FBs

   //Monitor TCP connection, if receive error has error above 80A1, then a comm error has occured and connection should be re-established
   IF #fbTRCV.STATUS >= 16#80A1 AND #bMQTT_Connected THEN
       #bTCP_Connected := FALSE;
       #bMQTT_Connected := FALSE;

       IF #iErrIndex > 10 THEN
           #iErrIndex := 1;
       END_IF;

       #iErrIndex := #iErrIndex + 1;

       //Reinit all subscribed topics
       FOR #i := 1 TO 20 BY 1 DO
           "dbMQTT_MessageBuffer".IncomingMessages.Message[#i].iStatus := 0;
       END_FOR;

       #iStatePublish := #ciPubError;
   END_IF;

   #fbTCON(REQ := (#iStatePublish = #ciEstablishTCP),
           ID := #TCON_Param.ID,
           CONNECT := #TCON_Param);

   #fbTDISCON(REQ := (#iStatePublish = #ciPubError),
              ID := #TCON_Param.ID);

   #fbTSEND(REQ := (#iStatePublish = #ciPubConnectSend) OR (#iStatePublish = #ciPubSend) OR (#iStateSubscribe = #ciSubSendSubscribe) OR (#iStateSubscribe = #ciSubSendPubAck),
            ID := #TCON_Param.ID,
            LEN := #uiSendLen,
            DATA := #byData);

   // Always listen after MQTT connected
   #fbTRCV(EN_R := (#bMQTT_Connected OR (#iStatePublish = #ciPubWaitConnack) OR (#iStatePublish = #ciPubWaitPubAck)),
           ID := #TCON_Param.ID,
           LEN := 1,
           DATA := #byData);

   // Only receive 1 byte at a time
   // Check that the last received message has been processed and all the relevent flags are reset
   IF (#fbTRCV.NDR AND NOT #bConAckReceived AND NOT #bPubAckReceived AND NOT #bSubAckReceived AND NOT #bPublishReceived AND NOT #bReceiveMessageComplete) THEN

       // Store recently received byte
       #byDataNewMessage[#iNewDataIndex] := #byData[1];

       // Check if we can calculate the total length of the message
       // Final byte of remaining length will have bit 7 set to 0
       // Enter conditional statement when you've reached final byte of remaining length
       IF #iNewDataIndex >= 2 AND (#byDataNewMessage[#iNewDataIndex] AND 2#10000000) = 0 AND #iReceiveMessageLength = 0 THEN
           #iReceiveLengthCalcIndex := 2;      // Set index to first byte of remaining length
           #iLen := 0;
           #multiplier := 1;
           REPEAT
               #byTemp := #byDataNewMessage[#iReceiveLengthCalcIndex];
               #iLen := #iLen + (#byTemp AND 2#01111111) * #multiplier;       // Add value encoded in byte to message length int
               #multiplier := #multiplier * 128;           // Scale up muliplier
               //TODO implement exception for length error
               #iReceiveLengthCalcIndex := #iReceiveLengthCalcIndex + 1;
           UNTIL ((#byTemp AND 2#1000000) = 0) END_REPEAT;
           #iReceiveMessageLength := #iLen;

       END_IF;

       // Continue Receiving bytes and incorporating them into byDataNewMessage until you've reached the end of the message
       IF (#iReceiveMessageLength + #iReceiveLengthCalcIndex - 1) = #iNewDataIndex THEN
           #bReceiveMessageComplete := TRUE;
       END_IF;

       #iNewDataIndex := #iNewDataIndex + 1;
   END_IF;

   //**********************************************************************************************************************
   // Reset all errors
   IF #bInResetError THEN
       #ERROR_MQTT.ConSendErr := FALSE;
       #ERROR_MQTT.ConSendTO := FALSE;
       #ERROR_MQTT.ConAckRcvErr := FALSE;
       #ERROR_MQTT.ConAckTO := FALSE;
       #ERROR_MQTT.ConAckIncReply := FALSE;
       #ERROR_MQTT.ConAckIncLen := FALSE;
       #ERROR_MQTT.ConAckUnacProt := FALSE;
       #ERROR_MQTT.ConAckIdRej := FALSE;
       #ERROR_MQTT.ConAckSerUn := FALSE;
       #ERROR_MQTT.ConAckUserPass := FALSE;
       #ERROR_MQTT.ConAckNotAut := FALSE;
       #ERROR_MQTT.ConAckUnknown := FALSE;
       #ERROR_MQTT.PubSendErr := FALSE;
       #ERROR_MQTT.PubSendTO := FALSE;
       #ERROR_MQTT.PubAckRcvErr := FALSE;
       #ERROR_MQTT.PubAckTO := FALSE;
       #ERROR_MQTT.PubAckIncReply := FALSE;
       #ERROR_MQTT.PubAckIncLen := FALSE;
       #ERROR_MQTT.PubAckPacketID := FALSE;
       #ERROR_MQTT.TcpErr := FALSE;
       #ERROR_MQTT.TcpTO := FALSE;
       #ERROR_MQTT.QueueOverflow := FALSE;
   END_IF;

   // At least one erorr is active - set output error flag
   #bOutError :=
   #ERROR_MQTT.ConSendErr OR
   #ERROR_MQTT.ConSendTO OR
   #ERROR_MQTT.ConAckRcvErr OR
   #ERROR_MQTT.ConAckTO OR
   #ERROR_MQTT.ConAckIncReply OR
   #ERROR_MQTT.ConAckIncLen OR
   #ERROR_MQTT.ConAckUnacProt OR
   #ERROR_MQTT.ConAckIdRej OR
   #ERROR_MQTT.ConAckSerUn OR
   #ERROR_MQTT.ConAckUserPass OR
   #ERROR_MQTT.ConAckNotAut OR
   #ERROR_MQTT.ConAckUnknown OR
   #ERROR_MQTT.PubSendErr OR
   #ERROR_MQTT.PubSendTO OR
   #ERROR_MQTT.PubAckRcvErr OR
   #ERROR_MQTT.PubAckTO OR
   #ERROR_MQTT.PubAckIncReply OR
   #ERROR_MQTT.PubAckIncLen OR
   #ERROR_MQTT.PubAckPacketID OR
   #ERROR_MQTT.SubSendErr OR
   #ERROR_MQTT.SubSendTimeout OR
   #ERROR_MQTT.SubAckIncReply OR
   #ERROR_MQTT.SubAckPacketID OR
   #ERROR_MQTT.SubAckRcvErr OR
   #ERROR_MQTT.SubAckTO OR
   #ERROR_MQTT.SubTopicNotFound OR
   #ERROR_MQTT.SubSendPubAckErr OR
   #ERROR_MQTT.SubSendPubAckTO OR
   #ERROR_MQTT.TcpErr OR
   #ERROR_MQTT.TcpTO OR
   #ERROR_MQTT.QueueOverflow;

   ENO := TRUE;
END_FUNCTION_BLOCK

FUNCTION "fcMQTT_SerializeMessageRaw" : Void   // FC3, SCL
{ S7_Optimized_Access := 'TRUE' }
VERSION : 0.1
   VAR_INPUT
      sInSerial : String;
      sInTopic : String;   // Topic to push data to
      sInVersion : String;   // Version of topic
      iInQoS : Int;   // Quality of Service needed
      Message : Variant;   // Data to be sent
   END_VAR
   VAR_OUTPUT
      bOutMessageSerialized : Bool;   // Set for one scan when message successfully entered into buffer
   END_VAR
   VAR_TEMP
      iTemp : Int;
      sTopicFull : String;   // Full topic name
      sTopicTemp1 : String;
      sTopicTemp2 : String;
      sVersion : String;
   END_VAR
BEGIN
   ///////////////////////////////////
   // Serialize Messages to be Sent //
   ///////////////////////////////////

   // Create Full Topic
   #sTopicTemp1 := CONCAT(IN1 := #sInSerial, IN2 := '/');
   #sTopicTemp2 := CONCAT(IN1 := #sTopicTemp1, IN2 := #sInTopic);
   #sTopicFull := CONCAT(IN1 := #sTopicTemp2, IN2 := #sInVersion);

   // Generate new global index to write    
   "dbMQTT_MessageBuffer".OutgoingMessages.iIndexWrite := "dbMQTT_MessageBuffer".OutgoingMessages.iIndexWrite + 1;

   // Check queue index at the end of the queue
   IF ("dbMQTT_MessageBuffer".OutgoingMessages.iIndexWrite > "dbMQTT_MessageBuffer".OutgoingMessages.iIndexMax) OR ("dbMQTT_MessageBuffer".OutgoingMessages.iIndexWrite <= 0) THEN
       "dbMQTT_MessageBuffer".OutgoingMessages.iIndexWrite := 1;
   END_IF;

   IF "dbMQTT_MessageBuffer".OutgoingMessages.Message["dbMQTT_MessageBuffer".OutgoingMessages.iIndexWrite].iStatus <> 0 THEN
       // Queue overfill detected
       "dbMQTT_MessageBuffer".OutgoingMessages.bErrorOverfill := true;
       #bOutMessageSerialized := FALSE;
   ELSE
       #bOutMessageSerialized := TRUE;
   END_IF;

   // Assign elements to the queue
   "dbMQTT_MessageBuffer".OutgoingMessages.Message["dbMQTT_MessageBuffer".OutgoingMessages.iIndexWrite].sTopic := #sTopicFull;
   "dbMQTT_MessageBuffer".OutgoingMessages.Message["dbMQTT_MessageBuffer".OutgoingMessages.iIndexWrite].iQoS := #iInQoS;

   // Reset message length parameter
   "dbMQTT_MessageBuffer".OutgoingMessages.Message["dbMQTT_MessageBuffer".OutgoingMessages.iIndexWrite].iMessageLength := 0;

   #iTemp := Serialize(SRC_VARIABLE:=#Message, DEST_ARRAY=>"dbMQTT_MessageBuffer".OutgoingMessages.Message["dbMQTT_MessageBuffer".OutgoingMessages.iIndexWrite].byValue,
                       POS:="dbMQTT_MessageBuffer".OutgoingMessages.Message["dbMQTT_MessageBuffer".OutgoingMessages.iIndexWrite].iMessageLength);


   // Update MQTT status
   "dbMQTT_MessageBuffer".OutgoingMessages.Message["dbMQTT_MessageBuffer".OutgoingMessages.iIndexWrite].iStatus := "ciReadyToPublish";

   ENO := TRUE;
END_FUNCTION

FUNCTION "fcMQTT_DeserializeMessageSubscribe" : Void   // FC5, SCL
{ S7_Optimized_Access := 'TRUE' }
VERSION : 0.1
   VAR_INPUT
      sInTopic : String;
      iInQoS : Int;
      iInBufferIndex : Int;
      sInSerial : String;
      sInVersion : String;
   END_VAR
   VAR_OUTPUT
      Message : Variant;
      bOutNewMessage : Bool;   // New message received, only active for one scan
   END_VAR
   VAR_TEMP
      iTemp : Int;
      iTemp2 : Int;
      diTemp : DInt;
      sTopicFull : String;
      sTopicTemp1 : String;
      sTopicTemp2 : String;
      sVersion : String;
   END_VAR
BEGIN
   // Create Full Topic
   #sTopicTemp1 := CONCAT(IN1 := #sInSerial, IN2 := '/');
   #sTopicTemp2 := CONCAT(IN1 := #sTopicTemp1, IN2 := #sInTopic);
   #sTopicFull := CONCAT(IN1 := #sTopicTemp2, IN2 := #sInVersion);

   //Check if subscribed
   IF ("dbMQTT_MessageBuffer".IncomingMessages.Message[#iInBufferIndex].iStatus = "ciSubDisabled") THEN
       "dbMQTT_MessageBuffer".IncomingMessages.Message[#iInBufferIndex].iStatus := "ciSubReadyToSub";
       "dbMQTT_MessageBuffer".IncomingMessages.Message[#iInBufferIndex].sTopic := #sTopicFull;
       "dbMQTT_MessageBuffer".IncomingMessages.Message[#iInBufferIndex].iQoS := #iInQoS;
   END_IF;

   // Deserialize received message
   IF ("dbMQTT_MessageBuffer".IncomingMessages.Message[#iInBufferIndex].iStatus = "ciSubMessageReceived") THEN
       #diTemp := 0;
       #iTemp := Deserialize(SRC_ARRAY := "dbMQTT_MessageBuffer".IncomingMessages.Message[#iInBufferIndex].byValue, DEST_VARIABLE => #Message, POS := #diTemp);
       "dbMQTT_MessageBuffer".IncomingMessages.Message[#iInBufferIndex].iStatus := "ciSubSubscribed";
       #bOutNewMessage := true;
   END_IF;
END_FUNCTION

// ===== library types =====

// folder: IOT

FUNCTION "fcMQTT_SerializeMessageJSON" : Void   // FC4, SCL
{ S7_Optimized_Access := 'TRUE' }
VERSION : 0.1
   VAR_INPUT
      sInTopic : String;   // Topic to push data to
      iInQoS : Int;   // Quality of Service needed
      Message : Variant;   // Data to be sent
   END_VAR
   VAR_OUTPUT
      bOutMessageSerialized : Bool;   // Set for one scan when message successfully entered into buffer
   END_VAR
   VAR_TEMP
      iTemp : Int;
   END_VAR
BEGIN




   // Generate new global index to write    
   "dbMQTT_MessageBuffer".OutgoingMessages.iIndexWrite := "dbMQTT_MessageBuffer".OutgoingMessages.iIndexWrite + 1;
   // Check queue index at the end of the queue
   IF ("dbMQTT_MessageBuffer".OutgoingMessages.iIndexWrite > "dbMQTT_MessageBuffer".OutgoingMessages.iIndexMax) OR ("dbMQTT_MessageBuffer".OutgoingMessages.iIndexWrite <= 0) THEN
       "dbMQTT_MessageBuffer".OutgoingMessages.iIndexWrite := 1;
   END_IF;

   IF "dbMQTT_MessageBuffer".OutgoingMessages.Message["dbMQTT_MessageBuffer".OutgoingMessages.iIndexWrite].iStatus <> 0 THEN
       // Queue overfill detected
       "dbMQTT_MessageBuffer".OutgoingMessages.bErrorOverfill := true;
       #bOutMessageSerialized := FALSE;
   ELSE
       #bOutMessageSerialized := TRUE;
   END_IF;

   // Assing element to the queue
   // TODO: BLKMOV instead?
   "dbMQTT_MessageBuffer".OutgoingMessages.Message["dbMQTT_MessageBuffer".OutgoingMessages.iIndexWrite].sTopic := #sInTopic;
   "dbMQTT_MessageBuffer".OutgoingMessages.Message["dbMQTT_MessageBuffer".OutgoingMessages.iIndexWrite].iQoS := #iInQoS;

   "dbMQTT_MessageBuffer".OutgoingMessages.Message["dbMQTT_MessageBuffer".OutgoingMessages.iIndexWrite].iMessageLength := 0;

   #iTemp := Serialize(SRC_VARIABLE:=#Message, DEST_ARRAY=>"dbMQTT_MessageBuffer".OutgoingMessages.Message["dbMQTT_MessageBuffer".OutgoingMessages.iIndexWrite].byValue,
                       POS:="dbMQTT_MessageBuffer".OutgoingMessages.Message["dbMQTT_MessageBuffer".OutgoingMessages.iIndexWrite].iMessageLength);


   // Update MQTT status
   "dbMQTT_MessageBuffer".OutgoingMessages.Message["dbMQTT_MessageBuffer".OutgoingMessages.iIndexWrite].iStatus := 10;

   ENO := TRUE;
END_FUNCTION